(* CODESYS project Cooking chamber.project

Project tree, tasks and I/O mapping:
  Device : L-force Panel Controller p300 Logic, Lenze, order no. LPC 1000, version 3.8.0.0
    application Application
      libraries: L_PLCDataManagerAccess, 3.0.0.0 (Lenze); L_PLCLoggingAccess, 3.3.0.0 (Lenze); L_Util, 3.3.0.0 (Lenze); CAA CiA 405, 3.5.3.0 (CAA Technical Workgroup)
      task MainTask (cyclic, interval t#10ms, priority 1) calls Main
      Programs/
        program Main [ST]
        Functions/
        Routines/
          program Controller [ST]
        Settings/
          program IOs [ST]
          program Timers [ST]
          program Process [ST]
      Variables/
        global variables Channels
        global variables Global
        global variables Settings
      Symbols/
        Symbols
    CANbus : CANbus, Lenze, version 2.0.0.0
      CANopen_Manager : CANopen_Manager, Lenze, version 3.12.0.0
          settings: Heartbeat Node ID = 63; Can Open Node ID = 63; ConfigVersion = 50659584
        EPM_S110 : EPM-S110, Lenze, order no. EPM-S110, version 1.12.0.0
            settings: General Options.Reset Node = FALSE; NODEIDSAVED = 1; SDO Timeout = 1000000; Explicit Deactivate PDOs = FALSE; PDO_Autoconfig = TRUE; EXPERTSETTINGS = TRUE; Emergency-General Parameters.Emergency enabled = FALSE; Emergency-General Parameters.Emergency COBID = 16#00000081; Settings.COBID = 16#00000201; Settings.Transmission Type = 16#FF; Settings.available PDO-Parameter.Inhibit Time available = FALSE; Settings.available PDO-Parameter.Event Timer available = FALSE; Settings.Inhibit Time = 0; Settings.Event Timer = 0; Generic COBID = '$NODEID+16#0200'; Settings.COBID = 16#00000181; Settings.Transmission Type = 16#FF; Settings.available PDO-Parameter.Inhibit Time available = TRUE; Settings.available PDO-Parameter.Event Timer available = TRUE; Settings.Inhibit Time = 0; Settings.Event Timer = 0; Generic COBID = '$NODEID+16#0180'; Setting /state digital Output : EPM_S302_DO8_DC24V_0_5A_02.Index = 16#6200; Setting /state digital Output : EPM_S302_DO8_DC24V_0_5A_02.Subindex = 16#01; Setting /state digital Output : EPM_S302_DO8_DC24V_0_5A_02.ObjectLength = 8; State digital input : EPM_S202_DI8_DC24V_00.Index = 16#6000; State digital input : EPM_S202_DI8_DC24V_00.Subindex = 16#01; State digital input : EPM_S202_DI8_DC24V_00.ObjectLength = 8; State digital input : EPM_S202_DI8_DC24V_01.Index = 16#6000; State digital input : EPM_S202_DI8_DC24V_01.Subindex = 16#02; State digital input : EPM_S202_DI8_DC24V_01.ObjectLength = 8; SDO List.Set Guardtime.Index = 16#100C; SDO List.Set Guardtime.Subindex = 16#00; SDO List.Set Guardtime.Value = 16#00000000; SDO List.Set Guardtime.Size = 16; SDO List.Set Guardtime.AbortIfError = FALSE; SDO List.Set Guardtime.JumpToLine = FALSE; SDO List.Set Guardtime.Line = 0; SDO List.Set Lifetime.Index = 16#100D; SDO List.Set Lifetime.Subindex = 16#00;
              SDO List.Set Lifetime.Value = 16#00000000; SDO List.Set Lifetime.Size = 8; SDO List.Set Lifetime.AbortIfError = FALSE; SDO List.Set Lifetime.JumpToLine = FALSE; SDO List.Set Lifetime.Line = 0; SDO List.Set Heartbeat Consumer.Index = 16#1016; SDO List.Set Heartbeat Consumer.Subindex = 16#01; SDO List.Set Heartbeat Consumer.Value = 0; SDO List.Set Heartbeat Consumer.Size = 32; SDO List.Set Heartbeat Consumer.AbortIfError = FALSE; SDO List.Set Heartbeat Consumer.JumpToLine = FALSE; SDO List.Set Heartbeat Consumer.Line = 0; SDO List.Set Heartbeat Consumer.Index = 16#1016; SDO List.Set Heartbeat Consumer.Subindex = 16#02; SDO List.Set Heartbeat Consumer.Value = 0; SDO List.Set Heartbeat Consumer.Size = 32; SDO List.Set Heartbeat Consumer.AbortIfError = FALSE; SDO List.Set Heartbeat Consumer.JumpToLine = FALSE; SDO List.Set Heartbeat Consumer.Line = 0; SDO List.Set Heartbeat Consumer.Index = 16#1016; SDO List.Set Heartbeat Consumer.Subindex = 16#03; SDO List.Set Heartbeat Consumer.Value = 0; SDO List.Set Heartbeat Consumer.Size = 32; SDO List.Set Heartbeat Consumer.AbortIfError = FALSE; SDO List.Set Heartbeat Consumer.JumpToLine = FALSE; SDO List.Set Heartbeat Consumer.Line = 0; SDO List.Set Heartbeat Consumer.Index = 16#1016; SDO List.Set Heartbeat Consumer.Subindex = 16#04; SDO List.Set Heartbeat Consumer.Value = 0; SDO List.Set Heartbeat Consumer.Size = 32; SDO List.Set Heartbeat Consumer.AbortIfError = FALSE; SDO List.Set Heartbeat Consumer.JumpToLine = FALSE; SDO List.Set Heartbeat Consumer.Line = 0; SDO List.Set Heartbeat Consumer.Index = 16#1016; SDO List.Set Heartbeat Consumer.Subindex = 16#05; SDO List.Set Heartbeat Consumer.Value = 0; SDO List.Set Heartbeat Consumer.Size = 32; SDO List.Set Heartbeat Consumer.AbortIfError = FALSE; SDO List.Set Heartbeat Consumer.JumpToLine = FALSE; SDO List.Set Heartbeat Consumer.Line = 0;
              SDO List.Set Heartbeat Producer.Index = 16#1017; SDO List.Set Heartbeat Producer.Subindex = 16#00; SDO List.Set Heartbeat Producer.Value = 16#00000000; SDO List.Set Heartbeat Producer.Size = 16; SDO List.Set Heartbeat Producer.AbortIfError = FALSE; SDO List.Set Heartbeat Producer.JumpToLine = FALSE; SDO List.Set Heartbeat Producer.Line = 0; SDO List.Disable PDO.Index = 16#1400; SDO List.Disable PDO.Subindex = 16#01; SDO List.Disable PDO.Value = 16#80000201; SDO List.Disable PDO.Size = 32; SDO List.Disable PDO.AbortIfError = FALSE; SDO List.Disable PDO.JumpToLine = FALSE; SDO List.Disable PDO.Line = 0; SDO List.Set transmission type.Index = 16#1400; SDO List.Set transmission type.Subindex = 16#02; SDO List.Set transmission type.Value = 16#FF; SDO List.Set transmission type.Size = 8; SDO List.Set transmission type.AbortIfError = FALSE; SDO List.Set transmission type.JumpToLine = FALSE; SDO List.Set transmission type.Line = 0; SDO List.Clear pdo mapping.Index = 16#1600; SDO List.Clear pdo mapping.Subindex = 16#00; SDO List.Clear pdo mapping.Value = 16#0; SDO List.Clear pdo mapping.Size = 8; SDO List.Clear pdo mapping.AbortIfError = FALSE; SDO List.Clear pdo mapping.JumpToLine = FALSE; SDO List.Clear pdo mapping.Line = 0; SDO List.Set Mapping.Index = 16#1600; SDO List.Set Mapping.Subindex = 16#01; SDO List.Set Mapping.Value = 16#62000108; SDO List.Set Mapping.Size = 32; SDO List.Set Mapping.AbortIfError = FALSE; SDO List.Set Mapping.JumpToLine = FALSE; SDO List.Set Mapping.Line = 0; SDO List.Set number of mappings.Index = 16#1600; SDO List.Set number of mappings.Subindex = 16#00; SDO List.Set number of mappings.Value = 16#01; SDO List.Set number of mappings.Size = 8; SDO List.Set number of mappings.AbortIfError = FALSE;
              SDO List.Set number of mappings.JumpToLine = FALSE; SDO List.Set number of mappings.Line = 0; SDO List.Set and enable COB-ID.Index = 16#1400; SDO List.Set and enable COB-ID.Subindex = 16#01; SDO List.Set and enable COB-ID.Value = 16#00000201; SDO List.Set and enable COB-ID.Size = 32; SDO List.Set and enable COB-ID.AbortIfError = FALSE; SDO List.Set and enable COB-ID.JumpToLine = FALSE; SDO List.Set and enable COB-ID.Line = 0; SDO List.Disable PDO.Index = 16#1800; SDO List.Disable PDO.Subindex = 16#01; SDO List.Disable PDO.Value = 16#80000181; SDO List.Disable PDO.Size = 32; SDO List.Disable PDO.AbortIfError = FALSE; SDO List.Disable PDO.JumpToLine = FALSE; SDO List.Disable PDO.Line = 0; SDO List.Set transmission type.Index = 16#1800; SDO List.Set transmission type.Subindex = 16#02; SDO List.Set transmission type.Value = 16#FF; SDO List.Set transmission type.Size = 8; SDO List.Set transmission type.AbortIfError = FALSE; SDO List.Set transmission type.JumpToLine = FALSE; SDO List.Set transmission type.Line = 0; SDO List.Set inhibit time.Index = 16#1800; SDO List.Set inhibit time.Subindex = 16#03; SDO List.Set inhibit time.Value = 16#0000; SDO List.Set inhibit time.Size = 16; SDO List.Set inhibit time.AbortIfError = FALSE; SDO List.Set inhibit time.JumpToLine = FALSE; SDO List.Set inhibit time.Line = 0; SDO List.Set event time.Index = 16#1800; SDO List.Set event time.Subindex = 16#05; SDO List.Set event time.Value = 16#0000; SDO List.Set event time.Size = 16; SDO List.Set event time.AbortIfError = FALSE; SDO List.Set event time.JumpToLine = FALSE; SDO List.Set event time.Line = 0; SDO List.Clear pdo mapping.Index = 16#1A00; SDO List.Clear pdo mapping.Subindex = 16#00; SDO List.Clear pdo mapping.Value = 16#0;
              SDO List.Clear pdo mapping.Size = 8; SDO List.Clear pdo mapping.AbortIfError = FALSE; SDO List.Clear pdo mapping.JumpToLine = FALSE; SDO List.Clear pdo mapping.Line = 0; SDO List.Set Mapping.Index = 16#1A00; SDO List.Set Mapping.Subindex = 16#01; SDO List.Set Mapping.Value = 16#60000108; SDO List.Set Mapping.Size = 32; SDO List.Set Mapping.AbortIfError = FALSE; SDO List.Set Mapping.JumpToLine = FALSE; SDO List.Set Mapping.Line = 0; SDO List.Set Mapping.Index = 16#1A00; SDO List.Set Mapping.Subindex = 16#02; SDO List.Set Mapping.Value = 16#60000208; SDO List.Set Mapping.Size = 32; SDO List.Set Mapping.AbortIfError = FALSE; SDO List.Set Mapping.JumpToLine = FALSE; SDO List.Set Mapping.Line = 0; SDO List.Set number of mappings.Index = 16#1A00; SDO List.Set number of mappings.Subindex = 16#00; SDO List.Set number of mappings.Value = 16#02; SDO List.Set number of mappings.Size = 8; SDO List.Set number of mappings.AbortIfError = FALSE; SDO List.Set number of mappings.JumpToLine = FALSE; SDO List.Set number of mappings.Line = 0; SDO List.Set and enable COB-ID.Index = 16#1800; SDO List.Set and enable COB-ID.Subindex = 16#01; SDO List.Set and enable COB-ID.Value = 16#00000181; SDO List.Set and enable COB-ID.Size = 32; SDO List.Set and enable COB-ID.AbortIfError = FALSE; SDO List.Set and enable COB-ID.JumpToLine = FALSE; SDO List.Set and enable COB-ID.Line = 0; ConfigVersion = 50659584
          EPM_S202_DI8_DC24V_00 : EPM-S202 DI8, DC24V, Lenze, order no. EPM-S202, version 1.12.0.0
              settings: Number of Params = 1; State digital input : EPM_S202_DI8_DC24V_00.Index = 16#6000; State digital input : EPM_S202_DI8_DC24V_00.Subindex = 16#01; State digital input : EPM_S202_DI8_DC24V_00.Startbit = 0; State digital input : EPM_S202_DI8_DC24V_00.Endbit = 7
              input  Application.Digital_input_channel_00[00] : BOOL  // State digital input : EPM_S202_DI8_DC24V_00.Bit0
              input  Application.Digital_input_channel_00[01] : BOOL  // State digital input : EPM_S202_DI8_DC24V_00.Bit1
              input  Application.Digital_input_channel_00[02] : BOOL  // State digital input : EPM_S202_DI8_DC24V_00.Bit2
              input  Application.Digital_input_channel_00[03] : BOOL  // State digital input : EPM_S202_DI8_DC24V_00.Bit3
              input  Application.Digital_input_channel_00[04] : BOOL  // State digital input : EPM_S202_DI8_DC24V_00.Bit4
              input  Application.Digital_input_channel_00[05] : BOOL  // State digital input : EPM_S202_DI8_DC24V_00.Bit5
              input  Application.Digital_input_channel_00[06] : BOOL  // State digital input : EPM_S202_DI8_DC24V_00.Bit6
              input  Application.Digital_input_channel_00[07] : BOOL  // State digital input : EPM_S202_DI8_DC24V_00.Bit7
              unmapped channels: State digital input : EPM_S202_DI8_DC24V_00
          EPM_S202_DI8_DC24V_01 : EPM-S202 DI8, DC24V, Lenze, order no. EPM-S202, version 1.12.0.0
              settings: Number of Params = 1; State digital input : EPM_S202_DI8_DC24V_01.Index = 16#6000; State digital input : EPM_S202_DI8_DC24V_01.Subindex = 16#02; State digital input : EPM_S202_DI8_DC24V_01.Startbit = 0; State digital input : EPM_S202_DI8_DC24V_01.Endbit = 7
              input  Application.Digital_input_channel_01[00] : BOOL  // State digital input : EPM_S202_DI8_DC24V_01.Bit0
              input  Application.Digital_input_channel_01[01] : BOOL  // State digital input : EPM_S202_DI8_DC24V_01.Bit1
              input  Application.Digital_input_channel_01[02] : BOOL  // State digital input : EPM_S202_DI8_DC24V_01.Bit2
              input  Application.Digital_input_channel_01[03] : BOOL  // State digital input : EPM_S202_DI8_DC24V_01.Bit3
              input  Application.Digital_input_channel_01[04] : BOOL  // State digital input : EPM_S202_DI8_DC24V_01.Bit4
              input  Application.Digital_input_channel_01[05] : BOOL  // State digital input : EPM_S202_DI8_DC24V_01.Bit5
              input  Application.Digital_input_channel_01[06] : BOOL  // State digital input : EPM_S202_DI8_DC24V_01.Bit6
              input  Application.Digital_input_channel_01[07] : BOOL  // State digital input : EPM_S202_DI8_DC24V_01.Bit7
              unmapped channels: State digital input : EPM_S202_DI8_DC24V_01
          EPM_S302_DO8_DC24V_0_5A_02 : EPM-S302 DO8, DC24V, 0,5A, Lenze, order no. EPM-S302, version 1.12.0.0
              settings: Number of Params = 1; Setting /state digital Output : EPM_S302_DO8_DC24V_0_5A_02.Index = 16#6200; Setting /state digital Output : EPM_S302_DO8_DC24V_0_5A_02.Subindex = 16#01; Setting /state digital Output : EPM_S302_DO8_DC24V_0_5A_02.Startbit = 0; Setting /state digital Output : EPM_S302_DO8_DC24V_0_5A_02.Endbit = 7
              output Application.Digital_output_channel_00[00] : BOOL  // Setting /state digital Output : EPM_S302_DO8_DC24V_0_5A_02.Bit0
              output Application.Digital_output_channel_00[01] : BOOL  // Setting /state digital Output : EPM_S302_DO8_DC24V_0_5A_02.Bit1
              output Application.Digital_output_channel_00[02] : BOOL  // Setting /state digital Output : EPM_S302_DO8_DC24V_0_5A_02.Bit2
              output Application.Digital_output_channel_00[03] : BOOL  // Setting /state digital Output : EPM_S302_DO8_DC24V_0_5A_02.Bit3
              output Application.Digital_output_channel_00[04] : BOOL  // Setting /state digital Output : EPM_S302_DO8_DC24V_0_5A_02.Bit4
              output Application.Digital_output_channel_00[05] : BOOL  // Setting /state digital Output : EPM_S302_DO8_DC24V_0_5A_02.Bit5
              output Application.Digital_output_channel_00[06] : BOOL  // Setting /state digital Output : EPM_S302_DO8_DC24V_0_5A_02.Bit6
              output Application.Digital_output_channel_00[07] : BOOL  // Setting /state digital Output : EPM_S302_DO8_DC24V_0_5A_02.Bit7
              unmapped channels: Setting /state digital Output : EPM_S302_DO8_DC24V_0_5A_02
*)

// Device/Application/Variables/Channels
VAR_GLOBAL
	
	// Analog input channel 00
		Analog_input_channel_00: ARRAY [00..07] OF LREAL;
	
	// Digital input channel 00
		Digital_input_channel_00: ARRAY [00..07] OF BOOL;
	
	// Digital input channel 01
		Digital_input_channel_01: ARRAY [00..07] OF BOOL;
	
	// Digital input channel 02
		Digital_input_channel_02: ARRAY [00..07] OF BOOL;
	
	// Digital output channel 00
		Digital_output_channel_00: ARRAY [00..07] OF BOOL;
	
	// Digital output channel 01
		Digital_output_channel_01: ARRAY [00..07] OF BOOL;
	
	// Digital output channel 02
		Digital_output_channel_02: ARRAY [00..07] OF BOOL;
	
	// Digital output channel 03
		Digital_output_channel_03: ARRAY [00..07] OF BOOL;
	
	// Digital output channel 04
		Digital_output_channel_04: ARRAY [00..07] OF BOOL;
	
	// Digital output channel 05
		Digital_output_channel_05: ARRAY [00..07] OF BOOL;

END_VAR

// Device/Application/Variables/Global
VAR_GLOBAL

	// Core product temperature sensor
		Core_temperature_sensor: ARRAY [00..02] OF REAL := [0, 0, 0];
	
	// Temperature sensor of the chamber
		Chamber_temperature_sensor: ARRAY [00..02] OF REAL := [0, 0, 0];
	
	// Core product temperature
		Core_temperature: ARRAY [00..02] OF REAL := [0, 0, 0];
	
	// Temperature chamber
		Chamber_temperature: ARRAY [00..02] OF REAL := [0, 0, 0];
		
	// Emergency control chamber
		Emergency_chamber: ARRAY [00..02] OF BOOL := [0, 0, 0];
	
	// Motor protection circuit
		Motor_protection: ARRAY [00..02] OF BOOL := [0, 0, 0];
	
	// Higher chimney closed
		Higher_chimney_closed: ARRAY [00..02] OF BOOL := [0, 0, 0];
	
	// Higher chimney open	
		Higher_chimney_open: ARRAY [00..02] OF BOOL := [0, 0, 0];
	
	// Lower chimney closed	
		Lower_chimney_closed: ARRAY [00..02] OF BOOL := [0, 0, 0];
	
	// Lower chimney open
		Lower_chimney_open: ARRAY [00..02] OF BOOL := [0, 0, 0];
	
	// Burner protection circuit
		Burner_protection: ARRAY [00..02] OF BOOL := [0, 0, 0];	
	
	// Activation motor
		Motor_activation: ARRAY [00..02, 00..10] OF BOOL := [0(0), 1(0), 2(0)];
	
	// Activation of the steam valve
		Steam_valve_activation: ARRAY [00..02] OF BOOL := [0, 0, 0];
	
	// Activation chimney
		Chimney_activation: ARRAY [00..02] OF BOOL := [0, 0, 0];
	
	// Activation smokehouse
		Smokehouse_activation: ARRAY [00..02] OF BOOL := [0, 0, 0];
	
	// Activation smokehouse
		Sound_activation: ARRAY [00..02] OF BOOL := [0, 0, 0];
	
	// Reset burner
		Burner_reset: ARRAY [00..02] OF BOOL := [0, 0, 0];

END_VAR

// Device/Application/Variables/Settings
VAR_GLOBAL PERSISTENT RETAIN
	
	// Core product temperature sensor offset
		Core_temperature_offset: ARRAY [00..02] OF REAL;
	
	// Temperature sensor of the chamber offset
		Chamber_temperature_offset: ARRAY [00..02] OF REAL;
		
END_VAR

// Device/Application/Programs/Main
PROGRAM Main
VAR
END_VAR

	
Controller();

IOs();
Process();

END_PROGRAM

// Device/Application/Programs/Routines/Controller
PROGRAM Controller
VAR
	merda00: INT := 100;
	merda01: INT;
	merda02: INT;
END_VAR

	
merda01 := merda01 + 1;

IF merda01 >= merda00 THEN
	
	merda02 := merda02 + 1;
	Motor_activation[00, 00] := TRUE;
	
	IF merda02 >= merda00 THEN
		
		merda01 := 0;
		merda02 := 0;
		Motor_activation[00, 00] := FALSE;
		
	END_IF
	
END_IF

END_PROGRAM

// Device/Application/Programs/Settings/IOs
PROGRAM IOs


// IO Configuration

	// Analog inputs
	
		// Core products temperature sensor
			Core_temperature_sensor[00] := Analog_input_channel_00[00];
			Core_temperature_sensor[01] := Analog_input_channel_00[01];
			Core_temperature_sensor[02] := Analog_input_channel_00[02];
	
		// Temperature sensor of the chambers
			Chamber_temperature_sensor[00] := Analog_input_channel_00[03];
			Chamber_temperature_sensor[01] := Analog_input_channel_00[04];
			Chamber_temperature_sensor[02] := Analog_input_channel_00[05];
			
	// Digital inputs
	
		// Emergency
			Emergency_chamber[00] := Digital_input_channel_00[00];
			Emergency_chamber[01] := Digital_input_channel_00[01];
			Emergency_chamber[02] := Digital_input_channel_00[02];
	
		// Protection of motors
			Motor_protection[00] := Digital_input_channel_00[03];
			Motor_protection[01] := Digital_input_channel_00[04];
			Motor_protection[02] := Digital_input_channel_00[05];
	
		// Higher chimneys closed
			Higher_chimney_closed[00] := Digital_input_channel_00[06];
			Higher_chimney_closed[01] := Digital_input_channel_00[07];
			Higher_chimney_closed[02] := Digital_input_channel_01[00];
	
		// Higher chimneys open
			Higher_chimney_open[00] := Digital_input_channel_01[01];
			Higher_chimney_open[01] := Digital_input_channel_01[02];
			Higher_chimney_open[02] := Digital_input_channel_01[03];
	
		// Lower chimneys closed
			Lower_chimney_closed[00] := Digital_input_channel_01[04];
			Lower_chimney_closed[01] := Digital_input_channel_01[05];
			Lower_chimney_closed[02] := Digital_input_channel_01[06];
	
		// Lower chimneys open
			Lower_chimney_open[00] := Digital_input_channel_01[07];
			Lower_chimney_open[01] := Digital_input_channel_02[00];
			Lower_chimney_open[02] := Digital_input_channel_02[01];
	
		// Burner
			Burner_protection[00] := Digital_input_channel_02[02];
			Burner_protection[01] := Digital_input_channel_02[03];
			Burner_protection[02] := Digital_input_channel_02[04];
			
	// Digital outputs
	
		// Activation motor
			Digital_output_channel_00[00] := Motor_activation[00, 00];
			Digital_output_channel_00[01] := Motor_activation[00, 01];
			Digital_output_channel_00[02] := Motor_activation[00, 02];
			Digital_output_channel_00[03] := Motor_activation[00, 03];
			Digital_output_channel_00[04] := Motor_activation[00, 04];
			Digital_output_channel_00[05] := Motor_activation[00, 05];
			Digital_output_channel_00[06] := Motor_activation[00, 06];
			Digital_output_channel_00[07] := Motor_activation[00, 07];
			Digital_output_channel_01[00] := Motor_activation[00, 08];
			Digital_output_channel_01[01] := Motor_activation[00, 09];
			Digital_output_channel_01[02] := Motor_activation[01, 00];
			Digital_output_channel_01[03] := Motor_activation[01, 01];
			Digital_output_channel_01[04] := Motor_activation[01, 02];
			Digital_output_channel_01[05] := Motor_activation[01, 03];
			Digital_output_channel_01[06] := Motor_activation[01, 04];
			Digital_output_channel_01[07] := Motor_activation[01, 05];
			Digital_output_channel_02[00] := Motor_activation[01, 06];
			Digital_output_channel_02[01] := Motor_activation[01, 07];
			Digital_output_channel_02[02] := Motor_activation[01, 08];
			Digital_output_channel_02[03] := Motor_activation[01, 09];
			Digital_output_channel_02[04] := Motor_activation[02, 00];
			Digital_output_channel_02[05] := Motor_activation[02, 01];
			Digital_output_channel_02[06] := Motor_activation[02, 02];
			Digital_output_channel_02[07] := Motor_activation[02, 03];
			Digital_output_channel_03[00] := Motor_activation[02, 04];
			Digital_output_channel_03[01] := Motor_activation[02, 05];
			Digital_output_channel_03[02] := Motor_activation[02, 06];
			Digital_output_channel_03[03] := Motor_activation[02, 07];
			Digital_output_channel_03[04] := Motor_activation[02, 08];
			Digital_output_channel_03[05] := Motor_activation[02, 09];
	
		// Activation of the steam valve
			Digital_output_channel_03[06] := Steam_valve_activation[00];
			Digital_output_channel_03[07] := Steam_valve_activation[01];
			Digital_output_channel_04[00] := Steam_valve_activation[02];
	
		// Drive chimney
			Digital_output_channel_04[01] := Chimney_activation[00];
			Digital_output_channel_04[02] := Chimney_activation[01];
			Digital_output_channel_04[03] := Chimney_activation[02];
	
		// Drive smokehouse
			Digital_output_channel_04[04] := Smokehouse_activation[00];
			Digital_output_channel_04[05] := Smokehouse_activation[01];
			Digital_output_channel_04[06] := Smokehouse_activation[02];
	
		// Drive sound
			Digital_output_channel_04[07] := Sound_activation[00];
			Digital_output_channel_05[00] := Sound_activation[01];
			Digital_output_channel_05[01] := Sound_activation[02];
	
		// Reset burner	
			Digital_output_channel_05[02] := Burner_reset[00];
			Digital_output_channel_05[03] := Burner_reset[01];
			Digital_output_channel_05[04] := Burner_reset[02];

END_PROGRAM

// Device/Application/Programs/Settings/Process
PROGRAM Process
VAR
END_VAR


// Calibration of the sensors

		// Core products temperature
			Core_temperature[00] := Core_temperature_sensor[00] + Core_temperature_offset[00];
			Core_temperature[01] := Core_temperature_sensor[01] + Core_temperature_offset[01];
			Core_temperature[02] := Core_temperature_sensor[02] + Core_temperature_offset[02];
	
		// Temperature chambers
			Chamber_temperature[00] := Chamber_temperature_sensor[00] + Chamber_temperature_offset[00];
			Chamber_temperature[01] := Chamber_temperature_sensor[01] + Chamber_temperature_offset[01];
			Chamber_temperature[02] := Chamber_temperature_sensor[02] + Chamber_temperature_offset[02];
	
// Digital output

END_PROGRAM

// Device/Application/Programs/Settings/Timers
PROGRAM Timers
VAR
END_VAR

END_PROGRAM
